FUNCTION TryConvert_DT_TO_LINT : BOOL
VAR_INPUT
	in : DT;
	out : REFERENCE TO LINT;
END_VAR

out := DT_TO_LINT(in);
TryConvert_DT_TO_LINT := TRUE;

END_FUNCTION

(* stored: Version 1.1.0.1, ProductVersion 3.1.4024.12
   POU TryConvert_DT_TO_LINT: Id {0eb2b8db-e9a8-41b9-b724-45840ef04ed7}, SpecialFunc None *)
